            // Weekend schedule
            IF currD = 0 OR currD = 6 THEN
                IF (wSchedWEHourStartF11_ <> wSchedWEHourEndF11_ OR wSchedWEMinStartF11_ <> wSchedWEMinEndF11_) THEN
                    // Schedule Unit ON
                    IF wSchedWEHourStartF11_ = currH AND wSchedWEMinStartF11_ = currM AND NOT bUnitTriggered THEN
                        bUnitTriggered := TRUE;
                        FOR i := 1 TO 22 DO
                            // Send command unit ON
                            IF bUnitF11_[i] THEN 
                                CASE i OF
                                    1: 
                                        //
                                        //FB_Bacnet.StartStopCommand_128.bEnWrite := TRUE;
                                        //FB_Bacnet.StartStopCommand_128.bVal := TRUE;
                                    2: 
                                        //
                                        //FB_Bacnet.StartStopCommand_129.bEnWrite := TRUE;
                                        //FB_Bacnet.StartStopCommand_129.bVal := TRUE;
                                    3: 
                                        //
                                        //FB_Bacnet.StartStopCommand_130.bEnWrite := TRUE;
                                        //FB_Bacnet.StartStopCommand_130.bVal := TRUE;
                                    4: 
                                        //
                                        //FB_Bacnet.StartStopCommand_131.bEnWrite := TRUE;
                                        //FB_Bacnet.StartStopCommand_131.bVal := TRUE;
                                    5: 
                                        //
                                        //FB_Bacnet.StartStopCommand_132.bEnWrite := TRUE;
                                        //FB_Bacnet.StartStopCommand_132.bVal := TRUE;
                                    6: 
                                        //
                                        //FB_Bacnet.StartStopCommand_133.bEnWrite := TRUE;
                                        //FB_Bacnet.StartStopCommand_133.bVal := TRUE;
                                    7: 
                                        //
                                        //FB_Bacnet.StartStopCommand_134.bEnWrite := TRUE;
                                        //FB_Bacnet.StartStopCommand_134.bVal := TRUE;
                                    8: 
                                        //
                                        //FB_Bacnet.StartStopCommand_135.bEnWrite := TRUE;
                                        //FB_Bacnet.StartStopCommand_135.bVal := TRUE;
                                    9: 
                                        //
                                        //FB_Bacnet.StartStopCommand_136.bEnWrite := TRUE;
                                        //FB_Bacnet.StartStopCommand_136.bVal := TRUE;
                                    10: 
                                        //
                                        //FB_Bacnet.StartStopCommand_137.bEnWrite := TRUE;
                                        //FB_Bacnet.StartStopCommand_137.bVal := TRUE;
                                    11: 
                                        //
                                        //FB_Bacnet.StartStopCommand_138.bEnWrite := TRUE;
                                        //FB_Bacnet.StartStopCommand_138.bVal := TRUE;
                                    12: 
                                        //
                                        //FB_Bacnet.StartStopCommand_139.bEnWrite := TRUE;
                                        //FB_Bacnet.StartStopCommand_139.bVal := TRUE;
                                    13: 
                                        //
                                        //FB_Bacnet.StartStopCommand_140.bEnWrite := TRUE;
                                        //FB_Bacnet.StartStopCommand_140.bVal := TRUE;
                                    14: 
                                        //
                                        //FB_Bacnet.StartStopCommand_141.bEnWrite := TRUE;
                                        //FB_Bacnet.StartStopCommand_141.bVal := TRUE;
                                    15: 
                                        //
                                        //FB_Bacnet.StartStopCommand_142.bEnWrite := TRUE;
                                        //FB_Bacnet.StartStopCommand_142.bVal := TRUE;
                                    16: 
                                        //
                                        //FB_Bacnet.StartStopCommand_143.bEnWrite := TRUE;
                                        //FB_Bacnet.StartStopCommand_143.bVal := TRUE;
                                    17: 
                                        
                                        FB_Bacnet.StartStopCommand_144.bEnWrite := TRUE;
                                        FB_Bacnet.StartStopCommand_144.bVal := TRUE;
                                    18: 
                                        //
                                        //FB_Bacnet.StartStopCommand_145.bEnWrite := TRUE;
                                        //FB_Bacnet.StartStopCommand_145.bVal := TRUE;
                                    19: 
                                        //
                                        //FB_Bacnet.StartStopCommand_146.bEnWrite := TRUE;
                                        //FB_Bacnet.StartStopCommand_146.bVal := TRUE;
                                    20: 
                                        //
                                        //FB_Bacnet.StartStopCommand_147.bEnWrite := TRUE;
                                        //FB_Bacnet.StartStopCommand_147.bVal := TRUE;
                                    21: 
                                        //
                                        //FB_Bacnet.StartStopCommand_148.bEnWrite := TRUE;
                                        //FB_Bacnet.StartStopCommand_148.bVal := TRUE;
                                    22: 
                                        
                                        FB_Bacnet_b.StartStopCommand_227.bEnWrite := TRUE;
                                        FB_Bacnet_b.StartStopCommand_227.bVal := TRUE;
                                END_CASE
                            END_IF
                        END_FOR
                    END_IF
                    // Schedule Unit OFF
                    IF wSchedWEHourEndF11_ = currH AND wSchedWEMinEndF11_ = currM AND NOT bUnitTriggered THEN
                        bUnitTriggered := TRUE;
                        FOR i := 1 TO 22 DO
                            // Send command unit OFF
                            IF bUnitF11_[i] THEN 
                                CASE i OF
                                    1: 
                                        //
                                        //FB_Bacnet.StartStopCommand_128.bEnWrite := TRUE;
                                        //FB_Bacnet.StartStopCommand_128.bVal := FALSE;
                                    2: 
                                        //
                                        //FB_Bacnet.StartStopCommand_129.bEnWrite := TRUE;
                                        //FB_Bacnet.StartStopCommand_129.bVal := FALSE;
                                    3: 
                                        //
                                        //FB_Bacnet.StartStopCommand_130.bEnWrite := TRUE;
                                        //FB_Bacnet.StartStopCommand_130.bVal := FALSE;
                                    4: 
                                        //
                                        //FB_Bacnet.StartStopCommand_131.bEnWrite := TRUE;
                                        //FB_Bacnet.StartStopCommand_131.bVal := FALSE;
                                    5: 
                                        //
                                        //FB_Bacnet.StartStopCommand_132.bEnWrite := TRUE;
                                        //FB_Bacnet.StartStopCommand_132.bVal := FALSE;
                                    6: 
                                        //
                                        //FB_Bacnet.StartStopCommand_133.bEnWrite := TRUE;
                                        //FB_Bacnet.StartStopCommand_133.bVal := FALSE;
                                    7: 
                                        //
                                        //FB_Bacnet.StartStopCommand_134.bEnWrite := TRUE;
                                        //FB_Bacnet.StartStopCommand_134.bVal := FALSE;
                                    8: 
                                        //
                                        //FB_Bacnet.StartStopCommand_135.bEnWrite := TRUE;
                                        //FB_Bacnet.StartStopCommand_135.bVal := FALSE;
                                    9: 
                                        //
                                        //FB_Bacnet.StartStopCommand_136.bEnWrite := TRUE;
                                        //FB_Bacnet.StartStopCommand_136.bVal := FALSE;
                                    10: 
                                        //
                                        //FB_Bacnet.StartStopCommand_137.bEnWrite := TRUE;
                                        //FB_Bacnet.StartStopCommand_137.bVal := FALSE;
                                    11: 
                                        //
                                        //FB_Bacnet.StartStopCommand_138.bEnWrite := TRUE;
                                        //FB_Bacnet.StartStopCommand_138.bVal := FALSE;
                                    12: 
                                        //
                                        //FB_Bacnet.StartStopCommand_139.bEnWrite := TRUE;
                                        //FB_Bacnet.StartStopCommand_139.bVal := FALSE;
                                    13: 
                                        //
                                        //FB_Bacnet.StartStopCommand_140.bEnWrite := TRUE;
                                        //FB_Bacnet.StartStopCommand_140.bVal := FALSE;
                                    14: 
                                        //
                                        //FB_Bacnet.StartStopCommand_141.bEnWrite := TRUE;
                                        //FB_Bacnet.StartStopCommand_141.bVal := FALSE;
                                    15: 
                                        //
                                        //FB_Bacnet.StartStopCommand_142.bEnWrite := TRUE;
                                        //FB_Bacnet.StartStopCommand_142.bVal := FALSE;
                                    16: 
                                        //
                                        //FB_Bacnet.StartStopCommand_143.bEnWrite := TRUE;
                                        //FB_Bacnet.StartStopCommand_143.bVal := FALSE;
                                    17: 
                                        //
                                        //FB_Bacnet.StartStopCommand_144.bEnWrite := TRUE;
                                        //FB_Bacnet.StartStopCommand_144.bVal := FALSE;
                                    18: 
                                        //
                                        //FB_Bacnet.StartStopCommand_145.bEnWrite := TRUE;
                                        //FB_Bacnet.StartStopCommand_145.bVal := FALSE;
                                    19: 
                                        //
                                        //FB_Bacnet.StartStopCommand_146.bEnWrite := TRUE;
                                        //FB_Bacnet.StartStopCommand_146.bVal := FALSE;
                                    20: 
                                        //
                                        //FB_Bacnet.StartStopCommand_147.bEnWrite := TRUE;
                                        //FB_Bacnet.StartStopCommand_147.bVal := FALSE;
                                    21: 
                                        //
                                        //FB_Bacnet.StartStopCommand_148.bEnWrite := TRUE;
                                        //FB_Bacnet.StartStopCommand_148.bVal := FALSE;
                                    22: 
                                        
                                        FB_Bacnet_b.StartStopCommand_227.bEnWrite := TRUE;
                                        FB_Bacnet_b.StartStopCommand_227.bVal := FALSE;
                                END_CASE
                            END_IF
                        END_FOR
                    END_IF
                END_IF
            END_IF
        END_IF

END_FUNCTION_BLOCK

// ---- POUs/FB_Scheduler/FB_Scheduler_F12.TcPOU

      FUNCTION_BLOCK FB_Scheduler_F12
      VAR_INPUT
          currH : WORD;
          currM : WORD;
          currD : WORD;
      END_VAR
      VAR_IN_OUT
          FB_Bacnet : FB_BACnet_DAIKIN_MasterStation_III_No_3;
      END_VAR
      VAR
          i : INT;
          bUnitTriggered : BOOL := FALSE; // New flag to track execution
          prevMinute : WORD := 0;        // New variable to track the previous minute
      END_VAR
      VAR PERSISTENT
          //scheduler var
          bEnSchedF12_ : BOOL := FALSE;
          wSchedWDHourStartF12_ : WORD; 
          wSchedWDMinStartF12_ : WORD; 
          wSchedWEHourStartF12_ : WORD; 
          wSchedWEMinStartF12_ : WORD;
          wSchedWDHourEndF12_ : WORD;
          wSchedWDMinEndF12_ : WORD;
          wSchedWEHourEndF12_ : WORD;
          wSchedWEMinEndF12_ : WORD;
          //unit var
          bUnitF12_ : ARRAY [1..24] OF BOOL;
      END_VAR


        // Reset trigger flag at minute change or at the exact scheduled time
        IF currM <> prevMinute OR 
           (currH = wSchedWDHourStartF12_ AND currM = wSchedWDMinStartF12_) OR 
           (currH = wSchedWDHourEndF12_ AND currM = wSchedWDMinEndF12_) THEN
            bUnitTriggered := FALSE;
            prevMinute := currM;
        END_IF

        // Unit Schedule Enable
        IF bEnSchedF12_ THEN
            // Weekday schedule
            IF currD >= 1 AND currD <= 5 THEN
                IF (wSchedWDHourStartF12_ <> wSchedWDHourEndF12_ OR wSchedWDMinStartF12_ <> wSchedWDMinEndF12_) THEN
                    // Schedule Unit ON
                    IF wSchedWDHourStartF12_ = currH AND wSchedWDMinStartF12_ = currM AND NOT bUnitTriggered THEN
                        bUnitTriggered := TRUE;
                        FOR i := 1 TO 24 DO
                            // Send command unit ON
                            IF bUnitF12_[i] THEN 
                                CASE i OF
                                    1: 
                                        //
                                        //FB_Bacnet.StartStopCommand_192.bEnWrite := TRUE;
                                        //FB_Bacnet.StartStopCommand_192.bVal := TRUE;
                                    2: 
                                        //
                                        //FB_Bacnet.StartStopCommand_193.bEnWrite := TRUE;
                                        //FB_Bacnet.StartStopCommand_193.bVal := TRUE;
                                    3: 
                                        //
                                        //FB_Bacnet.StartStopCommand_194.bEnWrite := TRUE;
                                        //FB_Bacnet.StartStopCommand_194.bVal := TRUE;
                                    4: 
                                        //
                                        //FB_Bacnet.StartStopCommand_195.bEnWrite := TRUE;
                                        //FB_Bacnet.StartStopCommand_195.bVal := TRUE;
                                    5: 
                                        //
                                        //FB_Bacnet.StartStopCommand_196.bEnWrite := TRUE;
                                        //FB_Bacnet.StartStopCommand_196.bVal := TRUE;
                                    6: 
                                        //
                                        //FB_Bacnet.StartStopCommand_197.bEnWrite := TRUE;
                                        //FB_Bacnet.StartStopCommand_197.bVal := TRUE;
                                    7: 
                                        //
                                        //FB_Bacnet.StartStopCommand_198.bEnWrite := TRUE;
                                        //FB_Bacnet.StartStopCommand_198.bVal := TRUE;
                                    8: 
                                        //
                                        //FB_Bacnet.StartStopCommand_199.bEnWrite := TRUE;
                                        //FB_Bacnet.StartStopCommand_199.bVal := TRUE;
                                    9: 
                                        //
                                        //FB_Bacnet.StartStopCommand_200.bEnWrite := TRUE;
                                        //FB_Bacnet.StartStopCommand_200.bVal := TRUE;
                                    10: 
                                        //
                                        //FB_Bacnet.StartStopCommand_201.bEnWrite := TRUE;
                                        //FB_Bacnet.StartStopCommand_201.bVal := TRUE;
                                    11: 
                                        //
                                        //FB_Bacnet.StartStopCommand_202.bEnWrite := TRUE;
                                        //FB_Bacnet.StartStopCommand_202.bVal := TRUE;
                                    12: 
                                        //
                                        //FB_Bacnet.StartStopCommand_203.bEnWrite := TRUE;
                                        //FB_Bacnet.StartStopCommand_203.bVal := TRUE;
                                    13: 
                                        //
                                        //FB_Bacnet.StartStopCommand_204.bEnWrite := TRUE;
                                        //FB_Bacnet.StartStopCommand_204.bVal := TRUE;
                                    14: 
                                        //
                                        //FB_Bacnet.StartStopCommand_205.bEnWrite := TRUE;
                                        //FB_Bacnet.StartStopCommand_205.bVal := TRUE;
                                    15: 
                                        //
                                        //FB_Bacnet.StartStopCommand_206.bEnWrite := TRUE;
                                        //FB_Bacnet.StartStopCommand_206.bVal := TRUE;
                                    16: 
                                        //
                                        //FB_Bacnet.StartStopCommand_207.bEnWrite := TRUE;
                                        //FB_Bacnet.StartStopCommand_207.bVal := TRUE;
                                    17: 
                                        //
                                        //FB_Bacnet.StartStopCommand_208.bEnWrite := TRUE;
                                        //FB_Bacnet.StartStopCommand_208.bVal := TRUE;
                                    18: 
                                        //
                                        //FB_Bacnet.StartStopCommand_209.bEnWrite := TRUE;
                                        //FB_Bacnet.StartStopCommand_209.bVal := TRUE;
                                    19: 
                                        //
                                        //FB_Bacnet.StartStopCommand_210.bEnWrite := TRUE;
                                        //FB_Bacnet.StartStopCommand_210.bVal := TRUE;
                                    20: 
                                        //
                                        //FB_Bacnet.StartStopCommand_211.bEnWrite := TRUE;
                                        //FB_Bacnet.StartStopCommand_211.bVal := TRUE;
                                    21: 
                                        //
                                        //FB_Bacnet.StartStopCommand_212.bEnWrite := TRUE;
                                        //FB_Bacnet.StartStopCommand_212.bVal := TRUE;
                                    22: 
                                        
                                        FB_Bacnet.StartStopCommand_224.bEnWrite := TRUE;
                                        FB_Bacnet.StartStopCommand_224.bVal := TRUE;
                                    23: 
                                        
                                        FB_Bacnet.StartStopCommand_225.bEnWrite := TRUE;
                                        FB_Bacnet.StartStopCommand_225.bVal := TRUE;
                                    24: 
                                        
                                        FB_Bacnet.StartStopCommand_226.bEnWrite := TRUE;
                                        FB_Bacnet.StartStopCommand_226.bVal := TRUE;
                                END_CASE
                            END_IF
                        END_FOR
                    END_IF
                    // Schedule Unit OFF
                    IF wSchedWDHourEndF12_ = currH AND wSchedWDMinEndF12_ = currM AND NOT bUnitTriggered THEN
                        bUnitTriggered := TRUE;
                        FOR i := 1 TO 24 DO
                            // Send command unit OFF
                            IF bUnitF12_[i] THEN 
                                CASE i OF
                                    1: 
                                        //
                                        //FB_Bacnet.StartStopCommand_192.bEnWrite := TRUE;
                                        //FB_Bacnet.StartStopCommand_192.bVal := FALSE;
                                    2: 
                                        //
                                        //FB_Bacnet.StartStopCommand_193.bEnWrite := TRUE;
                                        //FB_Bacnet.StartStopCommand_193.bVal := FALSE;
                                    3: 
                                        //
                                        //FB_Bacnet.StartStopCommand_194.bEnWrite := TRUE;
                                        //FB_Bacnet.StartStopCommand_194.bVal := FALSE;
                                    4: 
                                        //
                                        //FB_Bacnet.StartStopCommand_195.bEnWrite := TRUE;
                                        //FB_Bacnet.StartStopCommand_195.bVal := FALSE;
                                    5: 
                                        //
                                        //FB_Bacnet.StartStopCommand_196.bEnWrite := TRUE;
                                        //FB_Bacnet.StartStopCommand_196.bVal := FALSE;
                                    6: 
                                        //
                                        //FB_Bacnet.StartStopCommand_197.bEnWrite := TRUE;
                                        //FB_Bacnet.StartStopCommand_197.bVal := FALSE;
                                    7: 
                                        //
                                        //FB_Bacnet.StartStopCommand_198.bEnWrite := TRUE;
                                        //FB_Bacnet.StartStopCommand_198.bVal := FALSE;
                                    8: 
                                        //
                                        //FB_Bacnet.StartStopCommand_199.bEnWrite := TRUE;
                                        //FB_Bacnet.StartStopCommand_199.bVal := FALSE;
                                    9: 
                                        //
                                        //FB_Bacnet.StartStopCommand_200.bEnWrite := TRUE;
                                        //FB_Bacnet.StartStopCommand_200.bVal := FALSE;
                                    10: 
                                        //
                                        //FB_Bacnet.StartStopCommand_201.bEnWrite := TRUE;
                                        //FB_Bacnet.StartStopCommand_201.bVal := FALSE;
                                    11: 
                                        //
                                        //FB_Bacnet.StartStopCommand_202.bEnWrite := TRUE;
                                        //FB_Bacnet.StartStopCommand_202.bVal := FALSE;
                                    12: 
                                        //
                                        //FB_Bacnet.StartStopCommand_203.bEnWrite := TRUE;
                                        //FB_Bacnet.StartStopCommand_203.bVal := FALSE;
                                    13: 
                                        //
                                        //FB_Bacnet.StartStopCommand_204.bEnWrite := TRUE;
                                        //FB_Bacnet.StartStopCommand_204.bVal := FALSE;
                                    14: 
                                        //
                                        //FB_Bacnet.StartStopCommand_205.bEnWrite := TRUE;
                                        //FB_Bacnet.StartStopCommand_205.bVal := FALSE;
                                    15: 
                                        //
                                        //FB_Bacnet.StartStopCommand_206.bEnWrite := TRUE;
                                        //FB_Bacnet.StartStopCommand_206.bVal := FALSE;
                                    16: 
                                        //
                                        //FB_Bacnet.StartStopCommand_207.bEnWrite := TRUE;
                                        //FB_Bacnet.StartStopCommand_207.bVal := FALSE;
                                    17: 
                                        //
                                        //FB_Bacnet.StartStopCommand_208.bEnWrite := TRUE;
                                        //FB_Bacnet.StartStopCommand_208.bVal := FALSE;
                                    18: 
                                        //
                                        //FB_Bacnet.StartStopCommand_209.bEnWrite := TRUE;
                                        //FB_Bacnet.StartStopCommand_209.bVal := FALSE;
                                    19: 
                                        //
                                        //FB_Bacnet.StartStopCommand_210.bEnWrite := TRUE;
                                        //FB_Bacnet.StartStopCommand_210.bVal := FALSE;
                                    20: 
                                        //
                                        //FB_Bacnet.StartStopCommand_211.bEnWrite := TRUE;
                                        //FB_Bacnet.StartStopCommand_211.bVal := FALSE;
                                    21: 
                                        //
                                        //FB_Bacnet.StartStopCommand_212.bEnWrite := TRUE;
                                        //FB_Bacnet.StartStopCommand_212.bVal := FALSE;
                                    22: 
                                        
                                        FB_Bacnet.StartStopCommand_224.bEnWrite := TRUE;
                                        FB_Bacnet.StartStopCommand_224.bVal := FALSE;
                                    23: 
                                        
                                        FB_Bacnet.StartStopCommand_225.bEnWrite := TRUE;
                                        FB_Bacnet.StartStopCommand_225.bVal := FALSE;
                                    24: 
                                        
                                        FB_Bacnet.StartStopCommand_226.bEnWrite := TRUE;
                                        FB_Bacnet.StartStopCommand_226.bVal := FALSE;
                                END_CASE
                            END_IF
                        END_FOR
                    END_IF
                END_IF
            END_IF
        END_IF

        // Weekend schedule
        IF currD = 0 OR currD = 6 THEN
            IF (wSchedWEHourStartF12_ <> wSchedWEHourEndF12_ OR wSchedWEMinStartF12_ <> wSchedWEMinEndF12_) THEN
                // Schedule Unit ON
                IF wSchedWEHourStartF12_ = currH AND wSchedWEMinStartF12_ = currM AND NOT bUnitTriggered THEN
                    bUnitTriggered := TRUE;
                    FOR i := 1 TO 24 DO
                        // Send command unit ON
                        IF bUnitF12_[i] THEN 
                            CASE i OF
                                1: 
                                    //
                                    //FB_Bacnet.StartStopCommand_192.bEnWrite := TRUE;
                                    //FB_Bacnet.StartStopCommand_192.bVal := TRUE;
                                2: 
                                    //
                                    //FB_Bacnet.StartStopCommand_193.bEnWrite := TRUE;
                                    //FB_Bacnet.StartStopCommand_193.bVal := TRUE;
                                3: 
                                    //
                                    //FB_Bacnet.StartStopCommand_194.bEnWrite := TRUE;
                                    //FB_Bacnet.StartStopCommand_194.bVal := TRUE;
                                4: 
                                    //
                                    //FB_Bacnet.StartStopCommand_195.bEnWrite := TRUE;
                                    //FB_Bacnet.StartStopCommand_195.bVal := TRUE;
                                5: 
                                    //
                                    //FB_Bacnet.StartStopCommand_196.bEnWrite := TRUE;
                                    //FB_Bacnet.StartStopCommand_196.bVal := TRUE;
                                6: 
                                    //
                                    //FB_Bacnet.StartStopCommand_197.bEnWrite := TRUE;
                                    //FB_Bacnet.StartStopCommand_197.bVal := TRUE;
                                7: 
                                    //
                                    //FB_Bacnet.StartStopCommand_198.bEnWrite := TRUE;
                                    //FB_Bacnet.StartStopCommand_198.bVal := TRUE;
                                8: 
                                    //
                                    //FB_Bacnet.StartStopCommand_199.bEnWrite := TRUE;
                                    //FB_Bacnet.StartStopCommand_199.bVal := TRUE;
                                9: 
                                    //
                                    //FB_Bacnet.StartStopCommand_200.bEnWrite := TRUE;
                                    //FB_Bacnet.StartStopCommand_200.bVal := TRUE;
                                10: 
                                    //
                                    //FB_Bacnet.StartStopCommand_201.bEnWrite := TRUE;
                                    //FB_Bacnet.StartStopCommand_201.bVal := TRUE;
                                11: 
                                    //
                                    //FB_Bacnet.StartStopCommand_202.bEnWrite := TRUE;
                                    //FB_Bacnet.StartStopCommand_202.bVal := TRUE;
                                12: 
                                    //
                                    //FB_Bacnet.StartStopCommand_203.bEnWrite := TRUE;
                                    //FB_Bacnet.StartStopCommand_203.bVal := TRUE;
                                13: 
                                    //
                                    //FB_Bacnet.StartStopCommand_204.bEnWrite := TRUE;
                                    //FB_Bacnet.StartStopCommand_204.bVal := TRUE;
                                14: 
                                    //
                                    //FB_Bacnet.StartStopCommand_205.bEnWrite := TRUE;
                                    //FB_Bacnet.StartStopCommand_205.bVal := TRUE;
                                15: 
                                    //
                                    //FB_Bacnet.StartStopCommand_206.bEnWrite := TRUE;
                                    //FB_Bacnet.StartStopCommand_206.bVal := TRUE;
                                16: 
                                    //
                                    //FB_Bacnet.StartStopCommand_207.bEnWrite := TRUE;
                                    //FB_Bacnet.StartStopCommand_207.bVal := TRUE;
                                17: 
                                    //
                                    //FB_Bacnet.StartStopCommand_208.bEnWrite := TRUE;
                                    //FB_Bacnet.StartStopCommand_208.bVal := TRUE;
                                18: 
                                    //
                                    //FB_Bacnet.StartStopCommand_209.bEnWrite := TRUE;
                                    //FB_Bacnet.StartStopCommand_209.bVal := TRUE;
                                19: 
                                    //
                                    //FB_Bacnet.StartStopCommand_210.bEnWrite := TRUE;
                                    //FB_Bacnet.StartStopCommand_210.bVal := TRUE;
                                20: 
                                    //
                                    //FB_Bacnet.StartStopCommand_211.bEnWrite := TRUE;
                                    //FB_Bacnet.StartStopCommand_211.bVal := TRUE;
                                21: 
                                    //
                                    //FB_Bacnet.StartStopCommand_212.bEnWrite := TRUE;
                                    //FB_Bacnet.StartStopCommand_212.bVal := TRUE;
                                22: 
                                    
                                    FB_Bacnet.StartStopCommand_224.bEnWrite := TRUE;
                                    FB_Bacnet.StartStopCommand_224.bVal := TRUE;
                                23: 
                                    
                                    FB_Bacnet.StartStopCommand_225.bEnWrite := TRUE;
                                    FB_Bacnet.StartStopCommand_225.bVal := TRUE;
                                24: 
                                    
                                    FB_Bacnet.StartStopCommand_226.bEnWrite := TRUE;
                                    FB_Bacnet.StartStopCommand_226.bVal := TRUE;
                            END_CASE
                        END_IF
                    END_FOR
                END_IF
                // Schedule Unit OFF
                IF wSchedWEHourEndF12_ = currH AND wSchedWEMinEndF12_ = currM AND NOT bUnitTriggered THEN
                    bUnitTriggered := TRUE;
                    FOR i := 1 TO 24 DO
                        // Send command unit OFF
                        IF bUnitF12_[i] THEN 
                            CASE i OF
                                1: 
                                    //
                                    //FB_Bacnet.StartStopCommand_192.bEnWrite := TRUE;
                                    //FB_Bacnet.StartStopCommand_192.bVal := FALSE;
                                2: 
                                    //
                                    //FB_Bacnet.StartStopCommand_193.bEnWrite := TRUE;
                                    //FB_Bacnet.StartStopCommand_193.bVal := FALSE;
                                3: 
                                    //
                                    //FB_Bacnet.StartStopCommand_194.bEnWrite := TRUE;
                                    //FB_Bacnet.StartStopCommand_194.bVal := FALSE;
                                4: 
                                    //
                                    //FB_Bacnet.StartStopCommand_195.bEnWrite := TRUE;
                                    //FB_Bacnet.StartStopCommand_195.bVal := FALSE;
                                5: 
                                    //
                                    //FB_Bacnet.StartStopCommand_196.bEnWrite := TRUE;
                                    //FB_Bacnet.StartStopCommand_196.bVal := FALSE;
                                6: 
                                    //
                                    //FB_Bacnet.StartStopCommand_197.bEnWrite := TRUE;
                                    //FB_Bacnet.StartStopCommand_197.bVal := FALSE;
                                7: 
                                    //
                                    //FB_Bacnet.StartStopCommand_198.bEnWrite := TRUE;
                                    //FB_Bacnet.StartStopCommand_198.bVal := FALSE;
                                8: 
                                    //
                                    //FB_Bacnet.StartStopCommand_199.bEnWrite := TRUE;
                                    //FB_Bacnet.StartStopCommand_199.bVal := FALSE;
                                9: 
                                    //
                                    //FB_Bacnet.StartStopCommand_200.bEnWrite := TRUE;
                                    //FB_Bacnet.StartStopCommand_200.bVal := FALSE;
                                10: 
                                    //
                                    //FB_Bacnet.StartStopCommand_201.bEnWrite := TRUE;
                                    //FB_Bacnet.StartStopCommand_201.bVal := FALSE;
                                11: 
                                    //
                                    //FB_Bacnet.StartStopCommand_202.bEnWrite := TRUE;
                                    //FB_Bacnet.StartStopCommand_202.bVal := FALSE;
                                12: 
                                    //
                                    //FB_Bacnet.StartStopCommand_203.bEnWrite := TRUE;
                                    //FB_Bacnet.StartStopCommand_203.bVal := FALSE;
                                13: 
                                    //
                                    //FB_Bacnet.StartStopCommand_204.bEnWrite := TRUE;
                                    //FB_Bacnet.StartStopCommand_204.bVal := FALSE;
                                14: 
                                    //
                                    //FB_Bacnet.StartStopCommand_205.bEnWrite := TRUE;
                                    //FB_Bacnet.StartStopCommand_205.bVal := FALSE;
                                15: 
                                    //
                                    //FB_Bacnet.StartStopCommand_206.bEnWrite := TRUE;
                                    //FB_Bacnet.StartStopCommand_206.bVal := FALSE;
                                16: 
                                    //
                                    //FB_Bacnet.StartStopCommand_207.bEnWrite := TRUE;
                                    //FB_Bacnet.StartStopCommand_207.bVal := FALSE;
                                17: 
                                    //
                                    //FB_Bacnet.StartStopCommand_208.bEnWrite := TRUE;
                                    //FB_Bacnet.StartStopCommand_208.bVal := FALSE;
                                18: 
                                    //
                                    //FB_Bacnet.StartStopCommand_209.bEnWrite := TRUE;
                                    //FB_Bacnet.StartStopCommand_209.bVal := FALSE;
                                19: 
                                    //
                                    //FB_Bacnet.StartStopCommand_210.bEnWrite := TRUE;
                                    //FB_Bacnet.StartStopCommand_210.bVal := FALSE;
                                20: 
                                    //
                                    //FB_Bacnet.StartStopCommand_211.bEnWrite := TRUE;
                                    //FB_Bacnet.StartStopCommand_211.bVal := FALSE;
                                21: 
                                    //
                                    //FB_Bacnet.StartStopCommand_212.bEnWrite := TRUE;
                                    //FB_Bacnet.StartStopCommand_212.bVal := FALSE;
                                22: 
                                    
                                    FB_Bacnet.StartStopCommand_224.bEnWrite := TRUE;
                                    FB_Bacnet.StartStopCommand_224.bVal := FALSE;
                                23: 
                                    
                                    FB_Bacnet.StartStopCommand_225.bEnWrite := TRUE;
                                    FB_Bacnet.StartStopCommand_225.bVal := FALSE;
                                24: 
                                    
                                    FB_Bacnet.StartStopCommand_226.bEnWrite := TRUE;
                                    FB_Bacnet.StartStopCommand_226.bVal := FALSE;
                            END_CASE
                        END_IF
                    END_FOR
                END_IF
            END_IF
        END_IF

END_FUNCTION_BLOCK

// ---- POUs/FB_Scheduler/FB_Scheduler_F15.TcPOU

      FUNCTION_BLOCK FB_Scheduler_F15
      VAR_INPUT
          currH : WORD;
          currM : WORD;
          currD : WORD;
      END_VAR
      VAR_IN_OUT
          FB_Bacnet : FB_BACnet_DAIKIN_MasterStation_III_No_4;
          FB_Bacnet_b : FB_BACnet_DAIKIN_MasterStation_III_No_5;
      END_VAR
      VAR
          i : INT;
          bUnitTriggered : BOOL := FALSE; // New flag to track execution
          prevMinute : WORD := 0;        // New variable to track the previous minute
      END_VAR
      VAR PERSISTENT
          //scheduler var
          bEnSchedF15_ : BOOL := FALSE;
          wSchedWDHourStartF15_ : WORD; 
          wSchedWDMinStartF15_ : WORD; 
          wSchedWEHourStartF15_ : WORD; 
          wSchedWEMinStartF15_ : WORD;
          wSchedWDHourEndF15_ : WORD;
          wSchedWDMinEndF15_ : WORD;
          wSchedWEHourEndF15_ : WORD;
          wSchedWEMinEndF15_ : WORD;
          //unit var
          bUnitF15_ : ARRAY [1..23] OF BOOL;
      END_VAR


        // Reset trigger flag at minute change or at the exact scheduled time
        IF currM <> prevMinute OR 
           (currH = wSchedWDHourStartF15_ AND currM = wSchedWDMinStartF15_) OR 
           (currH = wSchedWDHourEndF15_ AND currM = wSchedWDMinEndF15_) THEN
            bUnitTriggered := FALSE;
            prevMinute := currM;
        END_IF

        // Unit Schedule Enable
        IF bEnSchedF15_ THEN
            // Weekday schedule
            IF currD >= 1 AND currD <= 5 THEN
                IF (wSchedWDHourStartF15_ <> wSchedWDHourEndF15_ OR wSchedWDMinStartF15_ <> wSchedWDMinEndF15_) THEN
                    // Schedule Unit ON
                    IF wSchedWDHourStartF15_ = currH AND wSchedWDMinStartF15_ = currM AND NOT bUnitTriggered THEN
                        bUnitTriggered := TRUE;
                        FOR i := 1 TO 23 DO
                            // Send command unit ON
                            IF bUnitF15_[i] THEN 
                                CASE i OF
                                    1: 
                                        
                                        FB_Bacnet.StartStopCommand_000.bEnWrite := TRUE;
                                        FB_Bacnet.StartStopCommand_000.bVal := TRUE;
                                    2: 
                                        
                                        FB_Bacnet.StartStopCommand_001.bEnWrite := TRUE;
                                        FB_Bacnet.StartStopCommand_001.bVal := TRUE;
                                    3: 
                                        
                                        FB_Bacnet.StartStopCommand_002.bEnWrite := TRUE;
                                        FB_Bacnet.StartStopCommand_002.bVal := TRUE;
                                    4: 
                                        
                                        FB_Bacnet.StartStopCommand_003.bEnWrite := TRUE;
                                        FB_Bacnet.StartStopCommand_003.bVal := TRUE;
                                    5: 
                                        
                                        FB_Bacnet.StartStopCommand_004.bEnWrite := TRUE;
                                        FB_Bacnet.StartStopCommand_004.bVal := TRUE;
                                    6: 
                                        
                                        FB_Bacnet.StartStopCommand_005.bEnWrite := TRUE;
                                        FB_Bacnet.StartStopCommand_005.bVal := TRUE;
                                    7: 
                                        
                                        FB_Bacnet.StartStopCommand_006.bEnWrite := TRUE;
                                        FB_Bacnet.StartStopCommand_006.bVal := TRUE;
                                    8: 
                                        
                                        FB_Bacnet.StartStopCommand_007.bEnWrite := TRUE;
                                        FB_Bacnet.StartStopCommand_007.bVal := TRUE;
                                    9: 
                                        
                                        FB_Bacnet.StartStopCommand_008.bEnWrite := TRUE;
                                        FB_Bacnet.StartStopCommand_008.bVal := TRUE;
                                    10: 
                                        
                                        FB_Bacnet.StartStopCommand_009.bEnWrite := TRUE;
                                        FB_Bacnet.StartStopCommand_009.bVal := TRUE;
                                    11: 
                                        
                                        FB_Bacnet.StartStopCommand_010.bEnWrite := TRUE;
                                        FB_Bacnet.StartStopCommand_010.bVal := TRUE;
                                    12: 
                                        
                                        FB_Bacnet.StartStopCommand_011.bEnWrite := TRUE;
                                        FB_Bacnet.StartStopCommand_011.bVal := TRUE;
                                    13: 
                                        
                                        FB_Bacnet.StartStopCommand_012.bEnWrite := TRUE;
                                        FB_Bacnet.StartStopCommand_012.bVal := TRUE;
                                    14: 
                                        
                                        FB_Bacnet.StartStopCommand_013.bEnWrite := TRUE;
                                        FB_Bacnet.StartStopCommand_013.bVal := TRUE;
                                    15: 
                                        
                                        FB_Bacnet.StartStopCommand_014.bEnWrite := TRUE;
                                        FB_Bacnet.StartStopCommand_014.bVal := TRUE;
                                    16: 
                                        
                                        FB_Bacnet.StartStopCommand_015.bEnWrite := TRUE;
                                        FB_Bacnet.StartStopCommand_015.bVal := TRUE;
                                    17: 
                                        
                                        FB_Bacnet.StartStopCommand_016.bEnWrite := TRUE;
                                        FB_Bacnet.StartStopCommand_016.bVal := TRUE;
                                    18: 
                                        
                                        FB_Bacnet.StartStopCommand_017.bEnWrite := TRUE;
                                        FB_Bacnet.StartStopCommand_017.bVal := TRUE;
                                    19: 
                                        
                                        FB_Bacnet.StartStopCommand_018.bEnWrite := TRUE;
                                        FB_Bacnet.StartStopCommand_018.bVal := TRUE;
                                    20: 
                                        
                                        FB_Bacnet.StartStopCommand_019.bEnWrite := TRUE;
                                        FB_Bacnet.StartStopCommand_019.bVal := TRUE;
                                    21: 
                                        
                                        FB_Bacnet.StartStopCommand_048.bEnWrite := TRUE;
                                        FB_Bacnet.StartStopCommand_048.bVal := TRUE;
                                    22: 
                                        
                                        FB_Bacnet_b.StartStopCommand_049.bEnWrite := TRUE;
                                        FB_Bacnet_b.StartStopCommand_049.bVal := TRUE;
                                    23: 
                                        
                                        FB_Bacnet_b.StartStopCommand_032.bEnWrite := TRUE;
                                        FB_Bacnet_b.StartStopCommand_032.bVal := TRUE;
                                END_CASE
                            END_IF
                        END_FOR
                    END_IF
                    // Schedule Unit OFF
                    IF wSchedWDHourEndF15_ = currH AND wSchedWDMinEndF15_ = currM AND NOT bUnitTriggered THEN
                        bUnitTriggered := TRUE;
                        FOR i := 1 TO 23 DO
                            // Send command unit OFF
                            IF bUnitF15_[i] THEN 
                                CASE i OF
                                    1: 
                                        
                                        FB_Bacnet.StartStopCommand_000.bEnWrite := TRUE;
                                        FB_Bacnet.StartStopCommand_000.bVal := FALSE;
                                    2: 
                                        
                                        FB_Bacnet.StartStopCommand_001.bEnWrite := TRUE;
                                        FB_Bacnet.StartStopCommand_001.bVal := FALSE;
                                    3: 
                                        
                                        FB_Bacnet.StartStopCommand_002.bEnWrite := TRUE;
                                        FB_Bacnet.StartStopCommand_002.bVal := FALSE;
                                    4: 
                                        
                                        FB_Bacnet.StartStopCommand_003.bEnWrite := TRUE;
                                        FB_Bacnet.StartStopCommand_003.bVal := FALSE;
                                    5: 
                                        
                                        FB_Bacnet.StartStopCommand_004.bEnWrite := TRUE;
                                        FB_Bacnet.StartStopCommand_004.bVal := FALSE;
                                    6: 
                                        
                                        FB_Bacnet.StartStopCommand_005.bEnWrite := TRUE;
                                        FB_Bacnet.StartStopCommand_005.bVal := FALSE;
                                    7: 
                                        
                                        FB_Bacnet.StartStopCommand_006.bEnWrite := TRUE;
                                        FB_Bacnet.StartStopCommand_006.bVal := FALSE;
                                    8: 
                                        
                                        FB_Bacnet.StartStopCommand_007.bEnWrite := TRUE;
                                        FB_Bacnet.StartStopCommand_007.bVal := FALSE;
                                    9: 
                                        
                                        FB_Bacnet.StartStopCommand_008.bEnWrite := TRUE;
                                        FB_Bacnet.StartStopCommand_008.bVal := FALSE;
                                    10: 
                                        
                                        FB_Bacnet.StartStopCommand_009.bEnWrite := TRUE;
                                        FB_Bacnet.StartStopCommand_009.bVal := FALSE;
                                    11: 
                                        
                                        FB_Bacnet.StartStopCommand_010.bEnWrite := TRUE;
                                        FB_Bacnet.StartStopCommand_010.bVal := FALSE;
                                    12: 
                                        
                                        FB_Bacnet.StartStopCommand_011.bEnWrite := TRUE;
                                        FB_Bacnet.StartStopCommand_011.bVal := FALSE;
                                    13: 
                                        
                                        FB_Bacnet.StartStopCommand_012.bEnWrite := TRUE;
                                        FB_Bacnet.StartStopCommand_012.bVal := FALSE;
                                    14: 
                                        
                                        FB_Bacnet.StartStopCommand_013.bEnWrite := TRUE;
                                        FB_Bacnet.StartStopCommand_013.bVal := FALSE;
                                    15: 
                                        
                                        FB_Bacnet.StartStopCommand_014.bEnWrite := TRUE;
                                        FB_Bacnet.StartStopCommand_014.bVal := FALSE;
                                    16: 
                                        
                                        FB_Bacnet.StartStopCommand_015.bEnWrite := TRUE;
                                        FB_Bacnet.StartStopCommand_015.bVal := FALSE;
                                    17: 
                                        
                                        FB_Bacnet.StartStopCommand_016.bEnWrite := TRUE;
                                        FB_Bacnet.StartStopCommand_016.bVal := FALSE;
                                    18: 
                                        
                                        FB_Bacnet.StartStopCommand_017.bEnWrite := TRUE;
                                        FB_Bacnet.StartStopCommand_017.bVal := FALSE;
                                    19: 
                                        
                                        FB_Bacnet.StartStopCommand_018.bEnWrite := TRUE;
                                        FB_Bacnet.StartStopCommand_018.bVal := FALSE;
                                    20: 
                                        
                                        FB_Bacnet.StartStopCommand_019.bEnWrite := TRUE;
                                        FB_Bacnet.StartStopCommand_019.bVal := FALSE;
                                    21: 
                                        
                                        FB_Bacnet.StartStopCommand_048.bEnWrite := TRUE;
                                        FB_Bacnet.StartStopCommand_048.bVal := FALSE;
                                    22: 
                                        
                                        FB_Bacnet_b.StartStopCommand_049.bEnWrite := TRUE;
                                        FB_Bacnet_b.StartStopCommand_049.bVal := FALSE;
                                    23: 
                                        
                                        FB_Bacnet_b.StartStopCommand_032.bEnWrite := TRUE;
                                        FB_Bacnet_b.StartStopCommand_032.bVal := FALSE;
                                END_CASE
                            END_IF
                        END_FOR
                    END_IF
                END_IF
            END_IF

            // Weekend schedule
            IF currD = 0 OR currD = 6 THEN
                IF (wSchedWEHourStartF15_ <> wSchedWEHourEndF15_ OR wSchedWEMinStartF15_ <> wSchedWEMinEndF15_) THEN
                    // Schedule Unit ON
                    IF wSchedWEHourStartF15_ = currH AND wSchedWEMinStartF15_ = currM AND NOT bUnitTriggered THEN
                        bUnitTriggered := TRUE;
                        FOR i := 1 TO 23 DO
                            // Send command unit ON
                            IF bUnitF15_[i] THEN 
                                CASE i OF
                                    1: 
                                        
                                        FB_Bacnet.StartStopCommand_000.bEnWrite := TRUE;
                                        FB_Bacnet.StartStopCommand_000.bVal := TRUE;
                                    2: 
                                        
                                        FB_Bacnet.StartStopCommand_001.bEnWrite := TRUE;
                                        FB_Bacnet.StartStopCommand_001.bVal := TRUE;
                                    3: 
                                        
                                        FB_Bacnet.StartStopCommand_002.bEnWrite := TRUE;
                                        FB_Bacnet.StartStopCommand_002.bVal := TRUE;
                                    4: 
                                        
                                        FB_Bacnet.StartStopCommand_003.bEnWrite := TRUE;
                                        FB_Bacnet.StartStopCommand_003.bVal := TRUE;
                                    5: 
                                        
                                        FB_Bacnet.StartStopCommand_004.bEnWrite := TRUE;
                                        FB_Bacnet.StartStopCommand_004.bVal := TRUE;
                                    6: 
                                        
                                        FB_Bacnet.StartStopCommand_005.bEnWrite := TRUE;
                                        FB_Bacnet.StartStopCommand_005.bVal := TRUE;
                                    7: 
                                        
                                        FB_Bacnet.StartStopCommand_006.bEnWrite := TRUE;
                                        FB_Bacnet.StartStopCommand_006.bVal := TRUE;
                                    8: 
                                        
                                        FB_Bacnet.StartStopCommand_007.bEnWrite := TRUE;
                                        FB_Bacnet.StartStopCommand_007.bVal := TRUE;
                                    9: 
                                        
                                        FB_Bacnet.StartStopCommand_008.bEnWrite := TRUE;
                                        FB_Bacnet.StartStopCommand_008.bVal := TRUE;
                                    10: 
                                        
                                        FB_Bacnet.StartStopCommand_009.bEnWrite := TRUE;
                                        FB_Bacnet.StartStopCommand_009.bVal := TRUE;
                                    11: 
                                        
                                        FB_Bacnet.StartStopCommand_010.bEnWrite := TRUE;
                                        FB_Bacnet.StartStopCommand_010.bVal := TRUE;
                                    12: 
                                        
                                        FB_Bacnet.StartStopCommand_011.bEnWrite := TRUE;
                                        FB_Bacnet.StartStopCommand_011.bVal := TRUE;
                                    13: 
                                        
                                        FB_Bacnet.StartStopCommand_012.bEnWrite := TRUE;
                                        FB_Bacnet.StartStopCommand_012.bVal := TRUE;
                                    14: 
                                        
                                        FB_Bacnet.StartStopCommand_013.bEnWrite := TRUE;
                                        FB_Bacnet.StartStopCommand_013.bVal := TRUE;
                                    15: 
                                        
                                        FB_Bacnet.StartStopCommand_014.bEnWrite := TRUE;
                                        FB_Bacnet.StartStopCommand_014.bVal := TRUE;
                                    16: 
                                        
                                        FB_Bacnet.StartStopCommand_015.bEnWrite := TRUE;
                                        FB_Bacnet.StartStopCommand_015.bVal := TRUE;
                                    17: 
                                        
                                        FB_Bacnet.StartStopCommand_016.bEnWrite := TRUE;
                                        FB_Bacnet.StartStopCommand_016.bVal := TRUE;
                                    18: 
                                        
                                        FB_Bacnet.StartStopCommand_017.bEnWrite := TRUE;
                                        FB_Bacnet.StartStopCommand_017.bVal := TRUE;
                                    19: 
                                        
                                        FB_Bacnet.StartStopCommand_018.bEnWrite := TRUE;
                                        FB_Bacnet.StartStopCommand_018.bVal := TRUE;
                                    20: 
                                        
                                        FB_Bacnet.StartStopCommand_019.bEnWrite := TRUE;
                                        FB_Bacnet.StartStopCommand_019.bVal := TRUE;
                                    21: 
                                        
                                        FB_Bacnet.StartStopCommand_048.bEnWrite := TRUE;
                                        FB_Bacnet.StartStopCommand_048.bVal := TRUE;
                                    22: 
                                        
                                        FB_Bacnet_b.StartStopCommand_049.bEnWrite := TRUE;
                                        FB_Bacnet_b.StartStopCommand_049.bVal := TRUE;
                                    23: 
                                        
                                        FB_Bacnet_b.StartStopCommand_032.bEnWrite := TRUE;
                                        FB_Bacnet_b.StartStopCommand_032.bVal := TRUE;
                                END_CASE
                            END_IF
                        END_FOR
                    END_IF
                    // Schedule Unit OFF
                    IF wSchedWEHourEndF15_ = currH AND wSchedWEMinEndF15_ = currM AND NOT bUnitTriggered THEN
                        bUnitTriggered := TRUE;
                        FOR i := 1 TO 23 DO
                            // Send command unit OFF
                            IF bUnitF15_[i] THEN 
                                CASE i OF
                                    1: 
                                        
                                        FB_Bacnet.StartStopCommand_000.bEnWrite := TRUE;
                                        FB_Bacnet.StartStopCommand_000.bVal := FALSE;
                                    2: 
                                        
                                        FB_Bacnet.StartStopCommand_001.bEnWrite := TRUE;
                                        FB_Bacnet.StartStopCommand_001.bVal := FALSE;
                                    3: 
                                        
                                        FB_Bacnet.StartStopCommand_002.bEnWrite := TRUE;
                                        FB_Bacnet.StartStopCommand_002.bVal := FALSE;
                                    4: 
                                        
                                        FB_Bacnet.StartStopCommand_003.bEnWrite := TRUE;
                                        FB_Bacnet.StartStopCommand_003.bVal := FALSE;
                                    5: 
                                        
                                        FB_Bacnet.StartStopCommand_004.bEnWrite := TRUE;
                                        FB_Bacnet.StartStopCommand_004.bVal := FALSE;
                                    6: 
                                        
                                        FB_Bacnet.StartStopCommand_005.bEnWrite := TRUE;
                                        FB_Bacnet.StartStopCommand_005.bVal := FALSE;
                                    7: 
                                        
                                        FB_Bacnet.StartStopCommand_006.bEnWrite := TRUE;
                                        FB_Bacnet.StartStopCommand_006.bVal := FALSE;
                                    8: 
                                        
                                        FB_Bacnet.StartStopCommand_007.bEnWrite := TRUE;
                                        FB_Bacnet.StartStopCommand_007.bVal := FALSE;
                                    9: 
                                        
                                        FB_Bacnet.StartStopCommand_008.bEnWrite := TRUE;
                                        FB_Bacnet.StartStopCommand_008.bVal := FALSE;
                                    10: 
                                        
                                        FB_Bacnet.StartStopCommand_009.bEnWrite := TRUE;
                                        FB_Bacnet.StartStopCommand_009.bVal := FALSE;
                                    11: 
                                        
                                        FB_Bacnet.StartStopCommand_010.bEnWrite := TRUE;
                                        FB_Bacnet.StartStopCommand_010.bVal := FALSE;
                                    12: 
                                        
                                        FB_Bacnet.StartStopCommand_011.bEnWrite := TRUE;
                                        FB_Bacnet.StartStopCommand_011.bVal := FALSE;
                                    13: 
                                        
                                        FB_Bacnet.StartStopCommand_012.bEnWrite := TRUE;
                                        FB_Bacnet.StartStopCommand_012.bVal := FALSE;
                                    14: 
                                        
                                        FB_Bacnet.StartStopCommand_013.bEnWrite := TRUE;
                                        FB_Bacnet.StartStopCommand_013.bVal := FALSE;
                                    15: 
                                        
                                        FB_Bacnet.StartStopCommand_014.bEnWrite := TRUE;
                                        FB_Bacnet.StartStopCommand_014.bVal := FALSE;
                                    16: 
                                        
                                        FB_Bacnet.StartStopCommand_015.bEnWrite := TRUE;
                                        FB_Bacnet.StartStopCommand_015.bVal := FALSE;
                                    17: 
                                        
                                        FB_Bacnet.StartStopCommand_016.bEnWrite := TRUE;
                                        FB_Bacnet.StartStopCommand_016.bVal := FALSE;
                                    18: 
                                        
                                        FB_Bacnet.StartStopCommand_017.bEnWrite := TRUE;
                                        FB_Bacnet.StartStopCommand_017.bVal := FALSE;
                                    19: 
                                        
                                        FB_Bacnet.StartStopCommand_018.bEnWrite := TRUE;
                                        FB_Bacnet.StartStopCommand_018.bVal := FALSE;
                                    20: 
                                        
                                        FB_Bacnet.StartStopCommand_019.bEnWrite := TRUE;
                                        FB_Bacnet.StartStopCommand_019.bVal := FALSE;
                                    21: 
                                        
                                        FB_Bacnet.StartStopCommand_048.bEnWrite := TRUE;
                                        FB_Bacnet.StartStopCommand_048.bVal := FALSE;
                                    22: 
                                        
                                        FB_Bacnet_b.StartStopCommand_049.bEnWrite := TRUE;
                                        FB_Bacnet_b.StartStopCommand_049.bVal := FALSE;
                                    23: 
                                        
                                        FB_Bacnet_b.StartStopCommand_032.bEnWrite := TRUE;
                                        FB_Bacnet_b.StartStopCommand_032.bVal := FALSE;
                                END_CASE
                            END_IF
                        END_FOR
                    END_IF
                END_IF
            END_IF
        END_IF

END_FUNCTION_BLOCK

// ---- POUs/FB_Scheduler/FB_Scheduler_F16.TcPOU

      FUNCTION_BLOCK FB_Scheduler_F16
      VAR_INPUT
          currH : WORD;
          currM : WORD;
          currD : WORD;
      END_VAR
      VAR_IN_OUT
          FB_Bacnet : FB_BACnet_DAIKIN_MasterStation_III_No_4;
          FB_Bacnet_b : FB_BACnet_DAIKIN_MasterStation_III_No_5;
      END_VAR
      VAR
          i : INT;
          bUnitTriggered : BOOL := FALSE; // New flag to track execution
          prevMinute : WORD := 0;        // New variable to track the previous minute
      END_VAR
      VAR PERSISTENT
          //scheduler var
          bEnSchedF16_ : BOOL := FALSE;
          wSchedWDHourStartF16_ : WORD; 
          wSchedWDMinStartF16_ : WORD; 
          wSchedWEHourStartF16_ : WORD; 
          wSchedWEMinStartF16_ : WORD;
          wSchedWDHourEndF16_ : WORD;
          wSchedWDMinEndF16_ : WORD;
          wSchedWEHourEndF16_ : WORD;
          wSchedWEMinEndF16_ : WORD;
          //unit var
          bUnitF16_ : ARRAY [1..21] OF BOOL;
      END_VAR


        // Reset trigger flag at minute change or at the exact scheduled time
        IF currM <> prevMinute OR 
           (currH = wSchedWDHourStartF16_ AND currM = wSchedWDMinStartF16_) OR 
           (currH = wSchedWDHourEndF16_ AND currM = wSchedWDMinEndF16_) THEN
            bUnitTriggered := FALSE;
            prevMinute := currM;
        END_IF

        // Unit Schedule Enable
        IF bEnSchedF16_ THEN
            // Weekday schedule
            IF currD >= 1 AND currD <= 5 THEN
                IF (wSchedWDHourStartF16_ <> wSchedWDHourEndF16_ OR wSchedWDMinStartF16_ <> wSchedWDMinEndF16_) THEN
                    // Schedule Unit ON
                    IF wSchedWDHourStartF16_ = currH AND wSchedWDMinStartF16_ = currM AND NOT bUnitTriggered THEN
                        bUnitTriggered := TRUE;
                        FOR i := 1 TO 21 DO
                            // Send command unit ON
                            IF bUnitF16_[i] THEN 
                                CASE i OF
                                    1: 
                                        
                                        FB_Bacnet.StartStopCommand_064.bEnWrite := TRUE;
                                        FB_Bacnet.StartStopCommand_064.bVal := TRUE;
                                    2: 
                                        
                                        FB_Bacnet.StartStopCommand_065.bEnWrite := TRUE;
                                        FB_Bacnet.StartStopCommand_065.bVal := TRUE;
                                    3: 
                                        
                                        FB_Bacnet.StartStopCommand_066.bEnWrite := TRUE;
                                        FB_Bacnet.StartStopCommand_066.bVal := TRUE;
                                    4: 
                                        
                                        FB_Bacnet.StartStopCommand_067.bEnWrite := TRUE;
                                        FB_Bacnet.StartStopCommand_067.bVal := TRUE;
                                    5: 
                                        
                                        FB_Bacnet.StartStopCommand_068.bEnWrite := TRUE;
                                        FB_Bacnet.StartStopCommand_068.bVal := TRUE;
                                    6: 
                                        
                                        FB_Bacnet.StartStopCommand_069.bEnWrite := TRUE;
                                        FB_Bacnet.StartStopCommand_069.bVal := TRUE;
                                    7: 
                                        
                                        FB_Bacnet.StartStopCommand_070.bEnWrite := TRUE;
                                        FB_Bacnet.StartStopCommand_070.bVal := TRUE;
                                    8: 
                                        
                                        FB_Bacnet.StartStopCommand_071.bEnWrite := TRUE;
                                        FB_Bacnet.StartStopCommand_071.bVal := TRUE;
                                    9: 
                                        
                                        FB_Bacnet.StartStopCommand_072.bEnWrite := TRUE;
                                        FB_Bacnet.StartStopCommand_072.bVal := TRUE;
                                    10: 
                                        
                                        FB_Bacnet.StartStopCommand_073.bEnWrite := TRUE;
                                        FB_Bacnet.StartStopCommand_073.bVal := TRUE;
                                    11: 
                                        
                                        FB_Bacnet.StartStopCommand_074.bEnWrite := TRUE;
                                        FB_Bacnet.StartStopCommand_074.bVal := TRUE;
                                    12: 
                                        
                                        FB_Bacnet.StartStopCommand_075.bEnWrite := TRUE;
                                        FB_Bacnet.StartStopCommand_075.bVal := TRUE;
                                    13: 
                                        
                                        FB_Bacnet.StartStopCommand_076.bEnWrite := TRUE;
                                        FB_Bacnet.StartStopCommand_076.bVal := TRUE;
                                    14: 
                                        
                                        FB_Bacnet.StartStopCommand_077.bEnWrite := TRUE;
                                        FB_Bacnet.StartStopCommand_077.bVal := TRUE;
                                    15: 
                                        
                                        FB_Bacnet.StartStopCommand_078.bEnWrite := TRUE;
                                        FB_Bacnet.StartStopCommand_078.bVal := TRUE;
                                    16: 
                                        
                                        FB_Bacnet.StartStopCommand_079.bEnWrite := TRUE;
                                        FB_Bacnet.StartStopCommand_079.bVal := TRUE;
                                    17: 
                                        
                                        FB_Bacnet.StartStopCommand_080.bEnWrite := TRUE;
                                        FB_Bacnet.StartStopCommand_080.bVal := TRUE;
                                    18: 
                                        
                                        FB_Bacnet.StartStopCommand_081.bEnWrite := TRUE;
                                        FB_Bacnet.StartStopCommand_081.bVal := TRUE;
                                    19: 
                                        
                                        FB_Bacnet.StartStopCommand_082.bEnWrite := TRUE;
                                        FB_Bacnet.StartStopCommand_082.bVal := TRUE;
                                    20: 
                                        
                                        FB_Bacnet.StartStopCommand_083.bEnWrite := TRUE;
                                        FB_Bacnet.StartStopCommand_083.bVal := TRUE;
                                    21: 
                                        
                                        FB_Bacnet_b.StartStopCommand_033.bEnWrite := TRUE;
                                        FB_Bacnet_b.StartStopCommand_033.bVal := TRUE;
                                END_CASE
                            END_IF
                        END_FOR
                    END_IF
                    // Schedule Unit OFF
                    IF wSchedWDHourEndF16_ = currH AND wSchedWDMinEndF16_ = currM AND NOT bUnitTriggered THEN
                        bUnitTriggered := TRUE;
                        FOR i := 1 TO 21 DO
                            // Send command unit OFF
                            IF bUnitF16_[i] THEN 
                                CASE i OF
                                    1: 
                                        
                                        FB_Bacnet.StartStopCommand_064.bEnWrite := TRUE;
                                        FB_Bacnet.StartStopCommand_064.bVal := FALSE;
                                    2: 
                                        
                                        FB_Bacnet.StartStopCommand_065.bEnWrite := TRUE;
                                        FB_Bacnet.StartStopCommand_065.bVal := FALSE;
                                    3: 
                                        
                                        FB_Bacnet.StartStopCommand_066.bEnWrite := TRUE;
                                        FB_Bacnet.StartStopCommand_066.bVal := FALSE;
                                    4: 
                                        
                                        FB_Bacnet.StartStopCommand_067.bEnWrite := TRUE;
                                        FB_Bacnet.StartStopCommand_067.bVal := FALSE;
                                    5: 
                                        
                                        FB_Bacnet.StartStopCommand_068.bEnWrite := TRUE;
                                        FB_Bacnet.StartStopCommand_068.bVal := FALSE;
                                    6: 
                                        
                                        FB_Bacnet.StartStopCommand_069.bEnWrite := TRUE;
                                        FB_Bacnet.StartStopCommand_069.bVal := FALSE;
                                    7: 
                                        
                                        FB_Bacnet.StartStopCommand_070.bEnWrite := TRUE;
                                        FB_Bacnet.StartStopCommand_070.bVal := FALSE;
                                    8: 
                                        
                                        FB_Bacnet.StartStopCommand_071.bEnWrite := TRUE;
                                        FB_Bacnet.StartStopCommand_071.bVal := FALSE;
                                    9: 
                                        
                                        FB_Bacnet.StartStopCommand_072.bEnWrite := TRUE;
                                        FB_Bacnet.StartStopCommand_072.bVal := FALSE;
                                    10: 
                                        
                                        FB_Bacnet.StartStopCommand_073.bEnWrite := TRUE;
                                        FB_Bacnet.StartStopCommand_073.bVal := FALSE;
                                    11: 
                                        
                                        FB_Bacnet.StartStopCommand_074.bEnWrite := TRUE;
                                        FB_Bacnet.StartStopCommand_074.bVal := FALSE;
                                    12: 
                                        
                                        FB_Bacnet.StartStopCommand_075.bEnWrite := TRUE;
                                        FB_Bacnet.StartStopCommand_075.bVal := FALSE;
                                    13: 
                                        
                                        FB_Bacnet.StartStopCommand_076.bEnWrite := TRUE;
                                        FB_Bacnet.StartStopCommand_076.bVal := FALSE;
                                    14: 
                                        
                                        FB_Bacnet.StartStopCommand_077.bEnWrite := TRUE;
                                        FB_Bacnet.StartStopCommand_077.bVal := FALSE;
                                    15: 
                                        
                                        FB_Bacnet.StartStopCommand_078.bEnWrite := TRUE;
                                        FB_Bacnet.StartStopCommand_078.bVal := FALSE;
                                    16: 
                                        
                                        FB_Bacnet.StartStopCommand_079.bEnWrite := TRUE;
                                        FB_Bacnet.StartStopCommand_079.bVal := FALSE;
                                    17: 
                                        
                                        FB_Bacnet.StartStopCommand_080.bEnWrite := TRUE;
                                        FB_Bacnet.StartStopCommand_080.bVal := FALSE;
                                    18: 
                                        
                                        FB_Bacnet.StartStopCommand_081.bEnWrite := TRUE;
                                        FB_Bacnet.StartStopCommand_081.bVal := FALSE;
                                    19: 
                                        
                                        FB_Bacnet.StartStopCommand_082.bEnWrite := TRUE;
                                        FB_Bacnet.StartStopCommand_082.bVal := FALSE;
                                    20: 
                                        
                                        FB_Bacnet.StartStopCommand_083.bEnWrite := TRUE;
                                        FB_Bacnet.StartStopCommand_083.bVal := FALSE;
                                    21: 
                                        
                                        FB_Bacnet_b.StartStopCommand_033.bEnWrite := TRUE;
                                        FB_Bacnet_b.StartStopCommand_033.bVal := FALSE;
                                END_CASE
                            END_IF
                        END_FOR
                    END_IF
                END_IF
            END_IF

            // Weekend schedule
            IF currD = 0 OR currD = 6 THEN
                IF (wSchedWEHourStartF16_ <> wSchedWEHourEndF16_ OR wSchedWEMinStartF16_ <> wSchedWEMinEndF16_) THEN
                    // Schedule Unit ON
                    IF wSchedWEHourStartF16_ = currH AND wSchedWEMinStartF16_ = currM AND NOT bUnitTriggered THEN
                        bUnitTriggered := TRUE;
                        FOR i := 1 TO 21 DO
                            // Send command unit ON
                            IF bUnitF16_[i] THEN 
                                CASE i OF
                                    1: 
                                        
                                        FB_Bacnet.StartStopCommand_064.bEnWrite := TRUE;
                                        FB_Bacnet.StartStopCommand_064.bVal := TRUE;
                                    2: 
                                        
                                        FB_Bacnet.StartStopCommand_065.bEnWrite := TRUE;
                                        FB_Bacnet.StartStopCommand_065.bVal := TRUE;
                                    3: 
                                        
                                        FB_Bacnet.StartStopCommand_066.bEnWrite := TRUE;
                                        FB_Bacnet.StartStopCommand_066.bVal := TRUE;
                                    4: 
                                        
                                        FB_Bacnet.StartStopCommand_067.bEnWrite := TRUE;
                                        FB_Bacnet.StartStopCommand_067.bVal := TRUE;
                                    5: 
                                        
                                        FB_Bacnet.StartStopCommand_068.bEnWrite := TRUE;
                                        FB_Bacnet.StartStopCommand_068.bVal := TRUE;
                                    6: 
                                        
                                        FB_Bacnet.StartStopCommand_069.bEnWrite := TRUE;
                                        FB_Bacnet.StartStopCommand_069.bVal := TRUE;
                                    7: 
                                        
                                        FB_Bacnet.StartStopCommand_070.bEnWrite := TRUE;
                                        FB_Bacnet.StartStopCommand_070.bVal := TRUE;
                                    8: 
                                        
                                        FB_Bacnet.StartStopCommand_071.bEnWrite := TRUE;
                                        FB_Bacnet.StartStopCommand_071.bVal := TRUE;
                                    9: 
                                        
                                        FB_Bacnet.StartStopCommand_072.bEnWrite := TRUE;
                                        FB_Bacnet.StartStopCommand_072.bVal := TRUE;
                                    10: 
                                        
                                        FB_Bacnet.StartStopCommand_073.bEnWrite := TRUE;
                                        FB_Bacnet.StartStopCommand_073.bVal := TRUE;
                                    11: 
                                        
                                        FB_Bacnet.StartStopCommand_074.bEnWrite := TRUE;
                                        FB_Bacnet.StartStopCommand_074.bVal := TRUE;
                                    12: 
                                        
                                        FB_Bacnet.StartStopCommand_075.bEnWrite := TRUE;
                                        FB_Bacnet.StartStopCommand_075.bVal := TRUE;
                                    13: 
                                        
                                        FB_Bacnet.StartStopCommand_076.bEnWrite := TRUE;
                                        FB_Bacnet.StartStopCommand_076.bVal := TRUE;
                                    14: 
                                        
                                        FB_Bacnet.StartStopCommand_077.bEnWrite := TRUE;
                                        FB_Bacnet.StartStopCommand_077.bVal := TRUE;
                                    15: 
                                        
                                        FB_Bacnet.StartStopCommand_078.bEnWrite := TRUE;
                                        FB_Bacnet.StartStopCommand_078.bVal := TRUE;
                                    16: 
                                        
                                        FB_Bacnet.StartStopCommand_079.bEnWrite := TRUE;
                                        FB_Bacnet.StartStopCommand_079.bVal := TRUE;
                                    17: 
                                        
                                        FB_Bacnet.StartStopCommand_080.bEnWrite := TRUE;
                                        FB_Bacnet.StartStopCommand_080.bVal := TRUE;
                                    18: 
                                        
                                        FB_Bacnet.StartStopCommand_081.bEnWrite := TRUE;
                                        FB_Bacnet.StartStopCommand_081.bVal := TRUE;
                                    19: 
                                        
                                        FB_Bacnet.StartStopCommand_082.bEnWrite := TRUE;
                                        FB_Bacnet.StartStopCommand_082.bVal := TRUE;
                                    20: 
                                        
                                        FB_Bacnet.StartStopCommand_083.bEnWrite := TRUE;
                                        FB_Bacnet.StartStopCommand_083.bVal := TRUE;
                                    21: 
                                        
                                        FB_Bacnet_b.StartStopCommand_033.bEnWrite := TRUE;
                                        FB_Bacnet_b.StartStopCommand_033.bVal := TRUE;
                                END_CASE
                            END_IF
                        END_FOR
                    END_IF
                    // Schedule Unit OFF
                    IF wSchedWEHourEndF16_ = currH AND wSchedWEMinEndF16_ = currM AND NOT bUnitTriggered THEN
                        bUnitTriggered := TRUE;
                        FOR i := 1 TO 21 DO
                            // Send command unit OFF
                            IF bUnitF16_[i] THEN 
                                CASE i OF
                                    1: 
                                        
                                        FB_Bacnet.StartStopCommand_064.bEnWrite := TRUE;
                                        FB_Bacnet.StartStopCommand_064.bVal := FALSE;
                                    2: 
                                        
                                        FB_Bacnet.StartStopCommand_065.bEnWrite := TRUE;
                                        FB_Bacnet.StartStopCommand_065.bVal := FALSE;
                                    3: 
                                        
                                        FB_Bacnet.StartStopCommand_066.bEnWrite := TRUE;
                                        FB_Bacnet.StartStopCommand_066.bVal := FALSE;
                                    4: 
                                        
                                        FB_Bacnet.StartStopCommand_067.bEnWrite := TRUE;
                                        FB_Bacnet.StartStopCommand_067.bVal := FALSE;
                                    5: 
                                        
                                        FB_Bacnet.StartStopCommand_068.bEnWrite := TRUE;
                                        FB_Bacnet.StartStopCommand_068.bVal := FALSE;
                                    6: 
                                        
                                        FB_Bacnet.StartStopCommand_069.bEnWrite := TRUE;
                                        FB_Bacnet.StartStopCommand_069.bVal := FALSE;
                                    7: 
                                        
                                        FB_Bacnet.StartStopCommand_070.bEnWrite := TRUE;
                                        FB_Bacnet.StartStopCommand_070.bVal := FALSE;
                                    8: 
                                        
                                        FB_Bacnet.StartStopCommand_071.bEnWrite := TRUE;
                                        FB_Bacnet.StartStopCommand_071.bVal := FALSE;
                                    9: 
                                        
                                        FB_Bacnet.StartStopCommand_072.bEnWrite := TRUE;
                                        FB_Bacnet.StartStopCommand_072.bVal := FALSE;
                                    10: 
                                        
                                        FB_Bacnet.StartStopCommand_073.bEnWrite := TRUE;
                                        FB_Bacnet.StartStopCommand_073.bVal := FALSE;
                                    11: 
                                        
                                        FB_Bacnet.StartStopCommand_074.bEnWrite := TRUE;
                                        FB_Bacnet.StartStopCommand_074.bVal := FALSE;
                                    12: 
                                        
                                        FB_Bacnet.StartStopCommand_075.bEnWrite := TRUE;
                                        FB_Bacnet.StartStopCommand_075.bVal := FALSE;
                                    13: 
                                        
                                        FB_Bacnet.StartStopCommand_076.bEnWrite := TRUE;
                                        FB_Bacnet.StartStopCommand_076.bVal := FALSE;
                                    14: 
                                        
                                        FB_Bacnet.StartStopCommand_077.bEnWrite := TRUE;
                                        FB_Bacnet.StartStopCommand_077.bVal := FALSE;
                                    15: 
                                        
                                        FB_Bacnet.StartStopCommand_078.bEnWrite := TRUE;
                                        FB_Bacnet.StartStopCommand_078.bVal := FALSE;
                                    16: 
                                        
                                        FB_Bacnet.StartStopCommand_079.bEnWrite := TRUE;
                                        FB_Bacnet.StartStopCommand_079.bVal := FALSE;
                                    17: 
                                        
                                        FB_Bacnet.StartStopCommand_080.bEnWrite := TRUE;
                                        FB_Bacnet.StartStopCommand_080.bVal := FALSE;
                                    18: 
                                        
                                        FB_Bacnet.StartStopCommand_081.bEnWrite := TRUE;
                                        FB_Bacnet.StartStopCommand_081.bVal := FALSE;
                                    19: 
                                        
                                        FB_Bacnet.StartStopCommand_082.bEnWrite := TRUE;
                                        FB_Bacnet.StartStopCommand_082.bVal := FALSE;
                                    20: 
                                        
                                        FB_Bacnet.StartStopCommand_083.bEnWrite := TRUE;
                                        FB_Bacnet.StartStopCommand_083.bVal := FALSE;
                                    21: 
                                        
                                        FB_Bacnet_b.StartStopCommand_033.bEnWrite := TRUE;
                                        FB_Bacnet_b.StartStopCommand_033.bVal := FALSE;
                                END_CASE
                            END_IF
                        END_FOR
                    END_IF
                END_IF
            END_IF
        END_IF

END_FUNCTION_BLOCK

// ---- POUs/FB_Scheduler/FB_Scheduler_F17.TcPOU

      FUNCTION_BLOCK FB_Scheduler_F17
      VAR_INPUT
          currH : WORD;
          currM : WORD;
          currD : WORD;
      END_VAR
      VAR_IN_OUT
          FB_Bacnet : FB_BACnet_DAIKIN_MasterStation_III_No_4;
          FB_Bacnet_b : FB_BACnet_DAIKIN_MasterStation_III_No_5;
      END_VAR
      VAR
          i : INT;
          bUnitTriggered : BOOL := FALSE; // New flag to track execution
          prevMinute : WORD := 0;        // New variable to track the previous minute
      END_VAR
      VAR PERSISTENT
          //scheduler var
          bEnSchedF17_ : BOOL := FALSE;
          wSchedWDHourStartF17_ : WORD; 
          wSchedWDMinStartF17_ : WORD; 
          wSchedWEHourStartF17_ : WORD; 
          wSchedWEMinStartF17_ : WORD;
          wSchedWDHourEndF17_ : WORD;
          wSchedWDMinEndF17_ : WORD;
          wSchedWEHourEndF17_ : WORD;
          wSchedWEMinEndF17_ : WORD;
          //unit var
          bUnitF17_ : ARRAY [1..21] OF BOOL;
      END_VAR


        // Reset trigger flag at minute change or at the exact scheduled time
        IF currM <> prevMinute OR 
           (currH = wSchedWDHourStartF17_ AND currM = wSchedWDMinStartF17_) OR 
           (currH = wSchedWDHourEndF17_ AND currM = wSchedWDMinEndF17_) THEN
            bUnitTriggered := FALSE;
            prevMinute := currM;
        END_IF

        // Unit Schedule Enable
        IF bEnSchedF17_ THEN
            // Weekday schedule
            IF currD >= 1 AND currD <= 5 THEN
                IF (wSchedWDHourStartF17_ <> wSchedWDHourEndF17_ OR wSchedWDMinStartF17_ <> wSchedWDMinEndF17_) THEN
                    // Schedule Unit ON
                    IF wSchedWDHourStartF17_ = currH AND wSchedWDMinStartF17_ = currM AND NOT bUnitTriggered THEN
                        bUnitTriggered := TRUE;
                        FOR i := 1 TO 21 DO
                            // Send command unit ON
                            IF bUnitF17_[i] THEN 
                                CASE i OF
                                    1: 
                                        
                                        FB_Bacnet.StartStopCommand_128.bEnWrite := TRUE;
                                        FB_Bacnet.StartStopCommand_128.bVal := TRUE;
                                    2: 
                                        
                                        FB_Bacnet.StartStopCommand_129.bEnWrite := TRUE;
                                        FB_Bacnet.StartStopCommand_129.bVal := TRUE;
                                    3: 
                                        
                                        FB_Bacnet.StartStopCommand_130.bEnWrite := TRUE;
                                        FB_Bacnet.StartStopCommand_130.bVal := TRUE;
                                    4: 
                                        
                                        FB_Bacnet.StartStopCommand_131.bEnWrite := TRUE;
                                        FB_Bacnet.StartStopCommand_131.bVal := TRUE;
                                    5: 
                                        
                                        FB_Bacnet.StartStopCommand_132.bEnWrite := TRUE;
                                        FB_Bacnet.StartStopCommand_132.bVal := TRUE;
                                    6: 
                                        
                                        FB_Bacnet.StartStopCommand_133.bEnWrite := TRUE;
                                        FB_Bacnet.StartStopCommand_133.bVal := TRUE;
                                    7: 
                                        
                                        FB_Bacnet.StartStopCommand_134.bEnWrite := TRUE;
                                        FB_Bacnet.StartStopCommand_134.bVal := TRUE;
                                    8: 
                                        
                                        FB_Bacnet.StartStopCommand_135.bEnWrite := TRUE;
                                        FB_Bacnet.StartStopCommand_135.bVal := TRUE;
                                    9: 
                                        
                                        FB_Bacnet.StartStopCommand_136.bEnWrite := TRUE;
                                        FB_Bacnet.StartStopCommand_136.bVal := TRUE;
                                    10: 
                                        
                                        FB_Bacnet.StartStopCommand_137.bEnWrite := TRUE;
                                        FB_Bacnet.StartStopCommand_137.bVal := TRUE;
                                    11: 
                                        
                                        FB_Bacnet.StartStopCommand_138.bEnWrite := TRUE;
                                        FB_Bacnet.StartStopCommand_138.bVal := TRUE;
                                    12: 
                                        
                                        FB_Bacnet.StartStopCommand_139.bEnWrite := TRUE;
                                        FB_Bacnet.StartStopCommand_139.bVal := TRUE;
                                    13: 
                                        
                                        FB_Bacnet.StartStopCommand_140.bEnWrite := TRUE;
                                        FB_Bacnet.StartStopCommand_140.bVal := TRUE;
                                    14: 
                                        
                                        FB_Bacnet.StartStopCommand_141.bEnWrite := TRUE;
                                        FB_Bacnet.StartStopCommand_141.bVal := TRUE;
                                    15: 
                                        
